FUNCTION_BLOCK SubMachine1 extends Composite
VAR
	component1					: Component;
	component2					: Component;
	childs						: ARRAY[1..NOOFCHILDS] OF IComposite := [component1,component2]; 
END_VAR
VAR CONSTANT
	NOOFCHILDS					: INT := 2;
END_VAR

METHOD logStatus
VAR
	sMessage				: STRING;		
	i						: DINT;
END_VAR
// Local status 
SUPER^.logStatus();

// Loop through childs
FOR i := 1 TO NOOFCHILDS DO
	IF childs[i]<>0 THEN
		childs[i].logStatus();
	END_IF
END_FOR
END_METHOD

END_FUNCTION_BLOCK

(* stored: Version 1.1.0.1, ProductVersion 3.1.4024.12
   POU SubMachine1: Id {044941f2-77fc-4748-bb6d-b1df11350035}, SpecialFunc None
   Method logStatus: Id {0438e7e8-ebfe-4cbc-8d52-20be17ea6aed} *)
